FUNCTION_BLOCK EL1008
VAR
	Channels : ARRAY [0..7] OF DigitalInputChannel;
END_VAR

METHOD PUBLIC GetDigitalInput : I_DigitalInput
VAR_INPUT
	channelNumber : INT;
END_VAR
GetDigitalInput := Channels[channelNumber];
END_METHOD

END_FUNCTION_BLOCK

(* stored: Version 1.1.0.1, ProductVersion 3.1.4024.5
   POU EL1008: Id {0cccfce6-a189-49df-b8cc-400af400ba61}, SpecialFunc None
   Method GetDigitalInput: Id {3b77e96f-55e6-4e9b-9d22-0d3911c37223} *)
